// TIA Portal V15.1 export
// export: Created 2024-05-17T05:38:38.2002518Z, ExportSetting WithDefaults, DisplayName Totally Integrated Automation Portal, DisplayVersion V15.1 Update 5, DisplayName TIA Portal Openness, DisplayVersion V15.1 Update 5, DisplayName SINAMICS Startdrive Advanced, DisplayVersion V15.1, DisplayName G130, G150, S120, S150, SINAMICS MV, S210, DisplayVersion V15.1, DisplayName G110M, G120, G120C, G120D, G120P, DisplayVersion V15.1, DisplayName STEP 7 Professional, DisplayVersion V15.1 Update 5, DisplayName STEP 7 Safety, DisplayVersion V15.1, DisplayName WinCC Professional, DisplayVersion V15.1 Update 5, DisplayName SIMATIC Visualization Architect, DisplayVersion V15.1
FUNCTION_BLOCK "LGBMotor2W1S-C"   // FB6612, FBD
TITLE = LGBMotor2W1S-C
{ S7_Optimized_Access := 'TRUE' }
AUTHOR : VCC
FAMILY : Actuator
VERSION : 0.1
// ============================================================================
// This "Motor-2Way-1Speed-Contactor" module is used in Applications when a Motor 
// 2 way - 1 speed equipped with contactors is needed.
// The module contains: a Motor loop equipped with 
// "1 Motor protection.
// "2 contactors (Set & Reset).
// "1 safety switch
// ============================================================================
// stored: AutoNumber false, IsIECCheckEnabled false, IsRetainMemResEnabled false, MemoryReserve 100, SetENOAutomatically False, UDAEnableTagReadback false
   VAR_INPUT
      I_EnableAlarm { ExternalAccessible := 'False'; ExternalVisible := 'False'; ExternalWritable := 'False'} : Bool;   // Enable Alarm
      I_MotorProtection { ExternalAccessible := 'False'; ExternalVisible := 'False'; ExternalWritable := 'False'} : Bool;   // Motor protection
      I_BrakeProtection { ExternalAccessible := 'False'; ExternalVisible := 'False'; ExternalWritable := 'False'} : Bool;   // Brake protection
      I_SafetySwitch { ExternalAccessible := 'False'; ExternalVisible := 'False'; ExternalWritable := 'False'} : Bool;   // Safety Switch
      I_SetMotorCmd { ExternalAccessible := 'False'; ExternalVisible := 'False'; ExternalWritable := 'False'} : Bool;   // Set Command from function after Interlock
      I_ResetMotorCmd { ExternalAccessible := 'False'; ExternalVisible := 'False'; ExternalWritable := 'False'} : Bool;   // Reset Command from function after Interlock
      I_AlarmResetPB { ExternalAccessible := 'False'; ExternalVisible := 'False'; ExternalWritable := 'False'} : Bool;   // Alarm Reset Pushbutton is Activated
      I_SafetyOk { ExternalAccessible := 'False'; ExternalVisible := 'False'; ExternalWritable := 'False'} : Bool;   // Safety Ok
      I_MotionStopOk { ExternalAccessible := 'False'; ExternalVisible := 'False'; ExternalWritable := 'False'} : Bool;   // Safety Ok / The motion stop is Ok
      I_BrakeReleased { ExternalAccessible := 'False'; ExternalVisible := 'False'; ExternalWritable := 'False'} : Bool;   // Brake Released or not used
   END_VAR
   VAR_OUTPUT
      O_MotorProtectionAlm { ExternalAccessible := 'False'; ExternalVisible := 'False'; ExternalWritable := 'False'} : Bool;   // Motor protection Alarm
      O_BrakeProtectionAlm { ExternalAccessible := 'False'; ExternalVisible := 'False'; ExternalWritable := 'False'} : Bool;   // Brake protection alarm
      O_SafetySwitchAlm { ExternalAccessible := 'False'; ExternalVisible := 'False'; ExternalWritable := 'False'} : Bool;   // Safety Switch Alarm
      O_MotionStopWarning { ExternalAccessible := 'False'; ExternalVisible := 'False'; ExternalWritable := 'False'} : Bool;   // Drive fault / Motion Stop warning
      O_BrakeFeedbackAlm { ExternalAccessible := 'False'; ExternalVisible := 'False'; ExternalWritable := 'False'} : Bool;   // Brake Feedback Alm
      O_SetContactor { ExternalAccessible := 'False'; ExternalVisible := 'False'; ExternalWritable := 'False'} : Bool;   // Set Contactor of Motor loop
      O_ResetContactor { ExternalAccessible := 'False'; ExternalVisible := 'False'; ExternalWritable := 'False'} : Bool;   // Reset Contactor of Motor loop
      O_ReleaseBrake { ExternalAccessible := 'False'; ExternalVisible := 'False'; ExternalWritable := 'False'} : Bool;   // Release Brake Contactor
      O_AlarmABCondition { ExternalAccessible := 'False'; ExternalVisible := 'False'; ExternalWritable := 'False'} : Bool;   // Alarm AB Condition
      O_Active { ExternalAccessible := 'False'; ExternalVisible := 'False'; ExternalWritable := 'False'} : Bool;   // Motor loop Active
   END_VAR
   VAR_IN_OUT
      IO_Modes : "Modes";
      IO_Alarm : "Alarm";
      H_HMI : "H_HMI";
      "H_GBMotor2W1S-C" : "H_GBMotor2W1S-C";   // Animation
      C_SafetySwNc { ExternalAccessible := 'False'; ExternalVisible := 'False'; ExternalWritable := 'False'} : Bool;   // Safety switch Normally closed
      C_SafetySwitchUsed { ExternalAccessible := 'False'; ExternalVisible := 'False'; ExternalWritable := 'False'} : Bool;   // Safety switch used
      C_MotorProtectionNc { ExternalAccessible := 'False'; ExternalVisible := 'False'; ExternalWritable := 'False'} : Bool;   // Motor Protection Normally closed
      C_MotorProtectionUsed { ExternalAccessible := 'False'; ExternalVisible := 'False'; ExternalWritable := 'False'} : Bool;   // Motor Protection used
      C_BrakeProtectionNc { ExternalAccessible := 'False'; ExternalVisible := 'False'; ExternalWritable := 'False'} : Bool;   // Motor Protection Normally closed / Brake Protection Normally closed
      C_BrakeProtectionUsed { ExternalAccessible := 'False'; ExternalVisible := 'False'; ExternalWritable := 'False'} : Bool;   // Brake Protection used / Motor Protection used
      C_BrakeUsed { ExternalAccessible := 'False'; ExternalVisible := 'False'; ExternalWritable := 'False'} : Bool;   // Brake Release Used
      C_MotionStopUsed { ExternalAccessible := 'False'; ExternalVisible := 'False'; ExternalWritable := 'False'} : Bool;   // Motion Stop used
   END_VAR
   VAR
      MotorProtectionAlm { ExternalAccessible := 'False'; ExternalVisible := 'False'; ExternalWritable := 'False'} : Bool;   // Motor protection Alarm
      BrakeProtectionAlm { ExternalAccessible := 'False'; ExternalVisible := 'False'; ExternalWritable := 'False'} : Bool;   // Brake protection alarm
      SafetySwitchAlm { ExternalAccessible := 'False'; ExternalVisible := 'False'; ExternalWritable := 'False'} : Bool;   // Safety Switch Alarm
      MotorProtectionAlmCond { ExternalAccessible := 'False'; ExternalVisible := 'False'; ExternalWritable := 'False'} : Bool;   // Motor protection Alarm condition
      BrakeProtectionAlmCond { ExternalAccessible := 'False'; ExternalVisible := 'False'; ExternalWritable := 'False'} : Bool;   // Brake protection alarm condition
      SafetySwitchAlmCond { ExternalAccessible := 'False'; ExternalVisible := 'False'; ExternalWritable := 'False'} : Bool;   // Safety Switch Alarm condition
      BrakeFeedbackAlm { ExternalAccessible := 'False'; ExternalVisible := 'False'; ExternalWritable := 'False'} : Bool;   // Safety Switch alarm / Safety Switch Alarm / BrakeFeedbackAlm
      MotionStopWarning { ExternalAccessible := 'False'; ExternalVisible := 'False'; ExternalWritable := 'False'} : Bool;   // Drive fault alarm / Motion Stop warning
      SetContactor { ExternalAccessible := 'False'; ExternalVisible := 'False'; ExternalWritable := 'False'} : Bool;   // Set Contactor of Motor loop
      ResetContactor { ExternalAccessible := 'False'; ExternalVisible := 'False'; ExternalWritable := 'False'} : Bool;   // Reset Contactor of Motor loop
      Active { ExternalAccessible := 'False'; ExternalVisible := 'False'; ExternalWritable := 'False'} : Bool;   // Motor loop Active
      _MotorProtection { ExternalAccessible := 'False'; ExternalVisible := 'False'; ExternalWritable := 'False'} : "L1AlarmMultiIn";   // FB
      _BrakeProtection { ExternalAccessible := 'False'; ExternalVisible := 'False'; ExternalWritable := 'False'} : "L1AlarmMultiIn";   // FB
      _SafetySwitch { ExternalAccessible := 'False'; ExternalVisible := 'False'; ExternalWritable := 'False'} : "L1AlarmMultiIn";   // FB
      _BrakeFeedback { ExternalAccessible := 'False'; ExternalVisible := 'False'; ExternalWritable := 'False'} : "L1AlarmMultiIn";   // FB
      _MotionStop { ExternalAccessible := 'False'; ExternalVisible := 'False'; ExternalWritable := 'False'} : "L1AlarmMultiIn";   // FB
      _TimeBrakeRelease { ExternalAccessible := 'False'; ExternalVisible := 'False'; ExternalWritable := 'False'} : TON_TIME;
      edge { ExternalAccessible := 'False'; ExternalVisible := 'False'; ExternalWritable := 'False'} : Array[0..1] of Bool;
   END_VAR
   VAR_TEMP   // added for the SCL form of the ladder/FBD networks
      _w1 : Bool;
      _w2 : Bool;
   END_VAR
BEGIN

REGION Network 1: ****2.1 - Enable Alarms **** Enable Brake Feedback Alarm
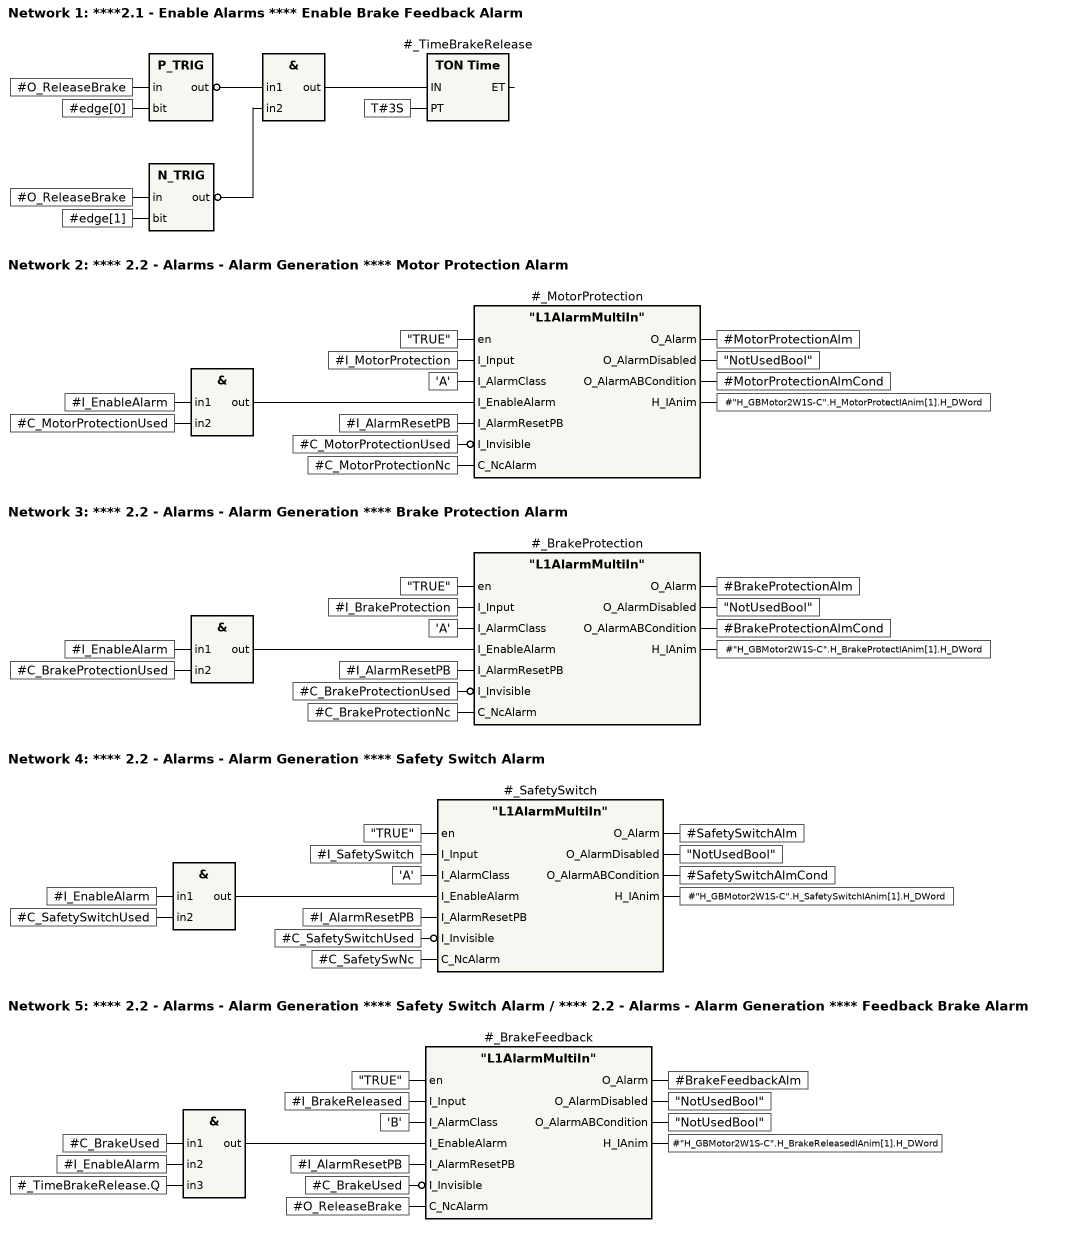
   #_w1 := #O_ReleaseBrake AND NOT #edge[0];   // rising edge
   #edge[0] := #O_ReleaseBrake;
   #_w2 := NOT #O_ReleaseBrake AND #edge[1];   // falling edge
   #edge[1] := #O_ReleaseBrake;
   #_TimeBrakeRelease(IN := NOT #_w1 AND NOT #_w2, PT := T#3S);   // TON
END_REGION

REGION Network 2: **** 2.2 - Alarms - Alarm Generation **** Motor Protection Alarm
   // Motor Protection Alarm
   IF "TRUE" THEN
       #_MotorProtection(I_Input := #I_MotorProtection,   // "L1AlarmMultiIn"
                         I_AlarmClass := 'A',
                         I_EnableAlarm := #I_EnableAlarm AND #C_MotorProtectionUsed,
                         I_AlarmResetPB := #I_AlarmResetPB,
                         I_Invisible := NOT #C_MotorProtectionUsed,
                         C_NcAlarm := #C_MotorProtectionNc,
                         O_Alarm => #MotorProtectionAlm,
                         O_AlarmDisabled => "NotUsedBool",
                         O_AlarmABCondition => #MotorProtectionAlmCond,
                         H_IAnim => #"H_GBMotor2W1S-C".H_MotorProtectIAnim[1].H_DWord);
   END_IF;
END_REGION

REGION Network 3: **** 2.2 - Alarms - Alarm Generation **** Brake Protection Alarm
   // Brake Protection Alarm
   IF "TRUE" THEN
       #_BrakeProtection(I_Input := #I_BrakeProtection,   // "L1AlarmMultiIn"
                         I_AlarmClass := 'A',
                         I_EnableAlarm := #I_EnableAlarm AND #C_BrakeProtectionUsed,
                         I_AlarmResetPB := #I_AlarmResetPB,
                         I_Invisible := NOT #C_BrakeProtectionUsed,
                         C_NcAlarm := #C_BrakeProtectionNc,
                         O_Alarm => #BrakeProtectionAlm,
                         O_AlarmDisabled => "NotUsedBool",
                         O_AlarmABCondition => #BrakeProtectionAlmCond,
                         H_IAnim => #"H_GBMotor2W1S-C".H_BrakeProtectIAnim[1].H_DWord);
   END_IF;
END_REGION

REGION Network 4: **** 2.2 - Alarms - Alarm Generation **** Safety Switch Alarm
   // Safety Switch Alarm
   IF "TRUE" THEN
       #_SafetySwitch(I_Input := #I_SafetySwitch,   // "L1AlarmMultiIn"
                      I_AlarmClass := 'A',
                      I_EnableAlarm := #I_EnableAlarm AND #C_SafetySwitchUsed,
                      I_AlarmResetPB := #I_AlarmResetPB,
                      I_Invisible := NOT #C_SafetySwitchUsed,
                      C_NcAlarm := #C_SafetySwNc,
                      O_Alarm => #SafetySwitchAlm,
                      O_AlarmDisabled => "NotUsedBool",
                      O_AlarmABCondition => #SafetySwitchAlmCond,
                      H_IAnim => #"H_GBMotor2W1S-C".H_SafetySwitchIAnim[1].H_DWord);
   END_IF;
END_REGION

REGION Network 5: **** 2.2 - Alarms - Alarm Generation **** Safety Switch Alarm / **** 2.2 - Alarms - Alarm Generation **** Feedback Brake Alarm
   // Safety Switch Alarm / Feedback Brake Alarm
   IF "TRUE" THEN
       #_BrakeFeedback(I_Input := #I_BrakeReleased,   // "L1AlarmMultiIn"
                       I_AlarmClass := 'B',
                       I_EnableAlarm := #C_BrakeUsed AND #I_EnableAlarm AND #_TimeBrakeRelease.Q,
                       I_AlarmResetPB := #I_AlarmResetPB,
                       I_Invisible := NOT #C_BrakeUsed,
                       C_NcAlarm := #O_ReleaseBrake,
                       O_Alarm => #BrakeFeedbackAlm,
                       O_AlarmDisabled => "NotUsedBool",
                       O_AlarmABCondition => "NotUsedBool",
                       H_IAnim => #"H_GBMotor2W1S-C".H_BrakeReleasedIAnim[1].H_DWord);
   END_IF;
END_REGION

REGION Network 6: **** 2.2 - Alarms - Alarm Generation **** MotionStop Warning
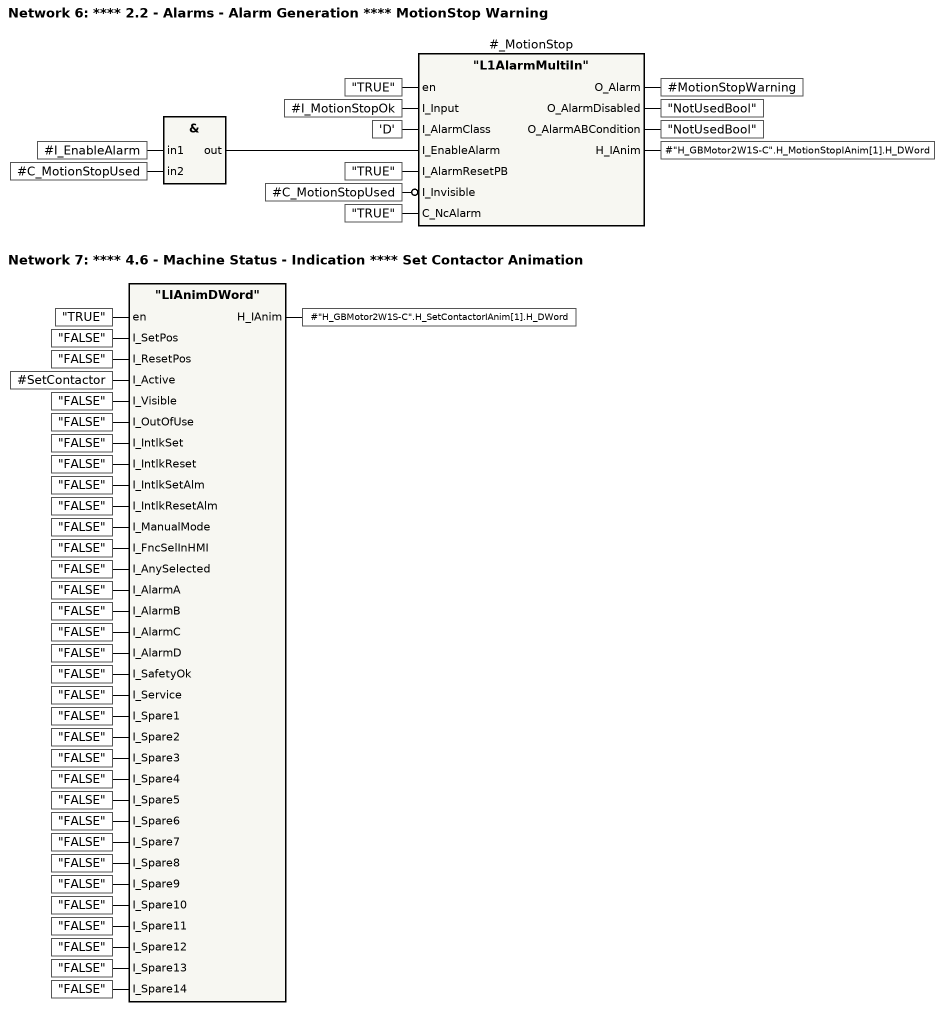
   IF "TRUE" THEN
       #_MotionStop(I_Input := #I_MotionStopOk,   // "L1AlarmMultiIn"
                    I_AlarmClass := 'D',
                    I_EnableAlarm := #I_EnableAlarm AND #C_MotionStopUsed,
                    I_AlarmResetPB := "TRUE",
                    I_Invisible := NOT #C_MotionStopUsed,
                    C_NcAlarm := "TRUE",
                    O_Alarm => #MotionStopWarning,
                    O_AlarmDisabled => "NotUsedBool",
                    O_AlarmABCondition => "NotUsedBool",
                    H_IAnim => #"H_GBMotor2W1S-C".H_MotionStopIAnim[1].H_DWord);
   END_IF;
END_REGION

REGION Network 7: **** 4.6 - Machine Status - Indication **** Set Contactor Animation
   // Set Contactor Animation
   IF "TRUE" THEN
       "LIAnimDWord"(I_SetPos := "FALSE",
                     I_ResetPos := "FALSE",
                     I_Active := #SetContactor,
                     I_Visible := "FALSE",
                     I_OutOfUse := "FALSE",
                     I_IntlkSet := "FALSE",
                     I_IntlkReset := "FALSE",
                     I_IntlkSetAlm := "FALSE",
                     I_IntlkResetAlm := "FALSE",
                     I_ManualMode := "FALSE",
                     I_FncSelInHMI := "FALSE",
                     I_AnySelected := "FALSE",
                     I_AlarmA := "FALSE",
                     I_AlarmB := "FALSE",
                     I_AlarmC := "FALSE",
                     I_AlarmD := "FALSE",
                     I_SafetyOk := "FALSE",
                     I_Service := "FALSE",
                     I_Spare1 := "FALSE",
                     I_Spare2 := "FALSE",
                     I_Spare3 := "FALSE",
                     I_Spare4 := "FALSE",
                     I_Spare5 := "FALSE",
                     I_Spare6 := "FALSE",
                     I_Spare7 := "FALSE",
                     I_Spare8 := "FALSE",
                     I_Spare9 := "FALSE",
                     I_Spare10 := "FALSE",
                     I_Spare11 := "FALSE",
                     I_Spare12 := "FALSE",
                     I_Spare13 := "FALSE",
                     I_Spare14 := "FALSE",
                     H_IAnim => #"H_GBMotor2W1S-C".H_SetContactorIAnim[1].H_DWord);
   END_IF;
END_REGION

REGION Network 8: **** 4.6 - Machine Status - Indication **** Reset Contactor Animation
   // Reset Contactor Animation
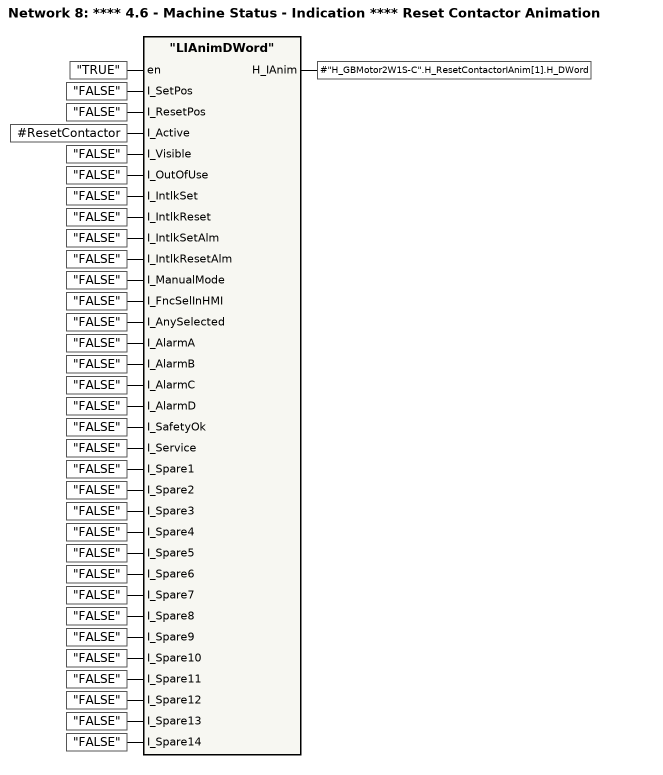
   IF "TRUE" THEN
       "LIAnimDWord"(I_SetPos := "FALSE",
                     I_ResetPos := "FALSE",
                     I_Active := #ResetContactor,
                     I_Visible := "FALSE",
                     I_OutOfUse := "FALSE",
                     I_IntlkSet := "FALSE",
                     I_IntlkReset := "FALSE",
                     I_IntlkSetAlm := "FALSE",
                     I_IntlkResetAlm := "FALSE",
                     I_ManualMode := "FALSE",
                     I_FncSelInHMI := "FALSE",
                     I_AnySelected := "FALSE",
                     I_AlarmA := "FALSE",
                     I_AlarmB := "FALSE",
                     I_AlarmC := "FALSE",
                     I_AlarmD := "FALSE",
                     I_SafetyOk := "FALSE",
                     I_Service := "FALSE",
                     I_Spare1 := "FALSE",
                     I_Spare2 := "FALSE",
                     I_Spare3 := "FALSE",
                     I_Spare4 := "FALSE",
                     I_Spare5 := "FALSE",
                     I_Spare6 := "FALSE",
                     I_Spare7 := "FALSE",
                     I_Spare8 := "FALSE",
                     I_Spare9 := "FALSE",
                     I_Spare10 := "FALSE",
                     I_Spare11 := "FALSE",
                     I_Spare12 := "FALSE",
                     I_Spare13 := "FALSE",
                     I_Spare14 := "FALSE",
                     H_IAnim => #"H_GBMotor2W1S-C".H_ResetContactorIAnim[1].H_DWord);
   END_IF;
END_REGION

REGION Network 9: **** 4.6 - Machine Status - Indication **** Reset Contactor Animation / **** 4.6 - Machine Status - Indication **** Release Brake Contactor Animation
   // Reset Contactor Animation
   // Release Brake Contactor Animation
   // Spare1 used to visualize the brake symbol on the contactor icon.
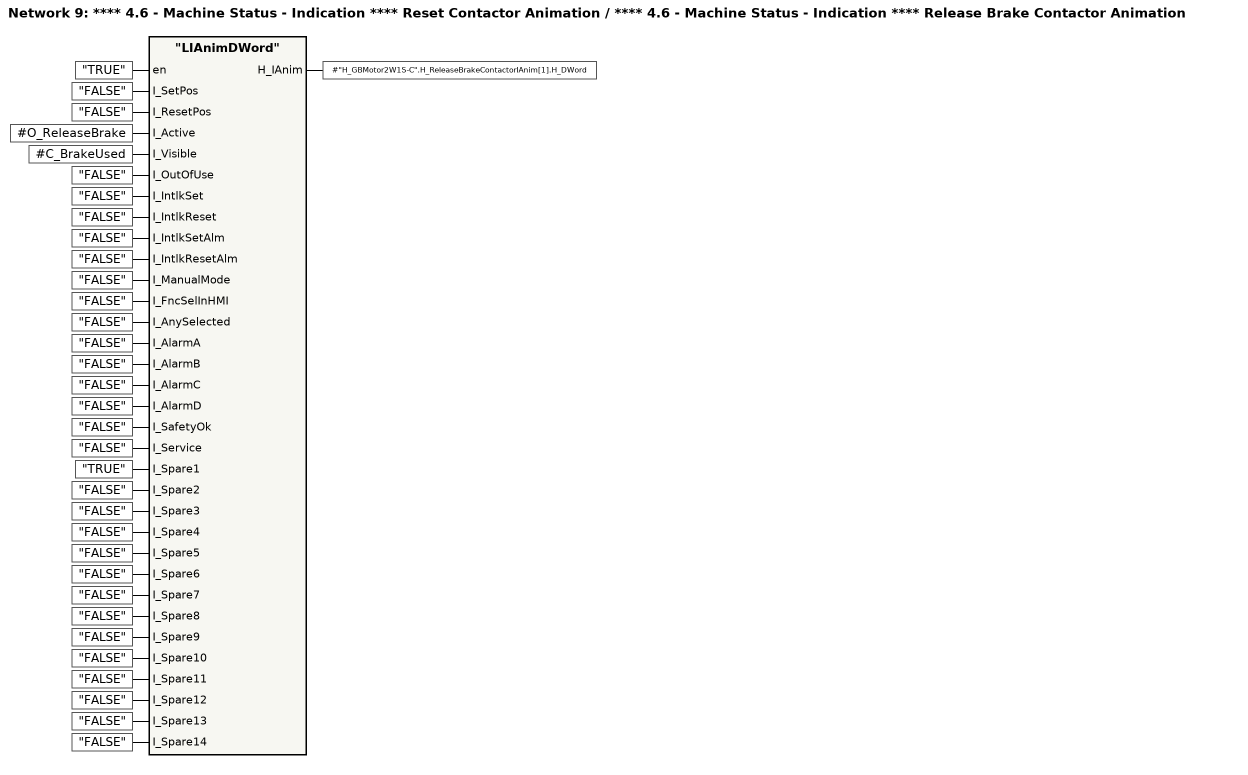
   IF "TRUE" THEN
       "LIAnimDWord"(I_SetPos := "FALSE",
                     I_ResetPos := "FALSE",
                     I_Active := #O_ReleaseBrake,
                     I_Visible := #C_BrakeUsed,
                     I_OutOfUse := "FALSE",
                     I_IntlkSet := "FALSE",
                     I_IntlkReset := "FALSE",
                     I_IntlkSetAlm := "FALSE",
                     I_IntlkResetAlm := "FALSE",
                     I_ManualMode := "FALSE",
                     I_FncSelInHMI := "FALSE",
                     I_AnySelected := "FALSE",
                     I_AlarmA := "FALSE",
                     I_AlarmB := "FALSE",
                     I_AlarmC := "FALSE",
                     I_AlarmD := "FALSE",
                     I_SafetyOk := "FALSE",
                     I_Service := "FALSE",
                     I_Spare1 := "TRUE",
                     I_Spare2 := "FALSE",
                     I_Spare3 := "FALSE",
                     I_Spare4 := "FALSE",
                     I_Spare5 := "FALSE",
                     I_Spare6 := "FALSE",
                     I_Spare7 := "FALSE",
                     I_Spare8 := "FALSE",
                     I_Spare9 := "FALSE",
                     I_Spare10 := "FALSE",
                     I_Spare11 := "FALSE",
                     I_Spare12 := "FALSE",
                     I_Spare13 := "FALSE",
                     I_Spare14 := "FALSE",
                     H_IAnim => #"H_GBMotor2W1S-C".H_ReleaseBrakeContactorIAnim[1].H_DWord);
   END_IF;
END_REGION

REGION Network 10: **** 4.6 - Machine Status - Indication **** Motor Icon Animation
   // Motor Animation
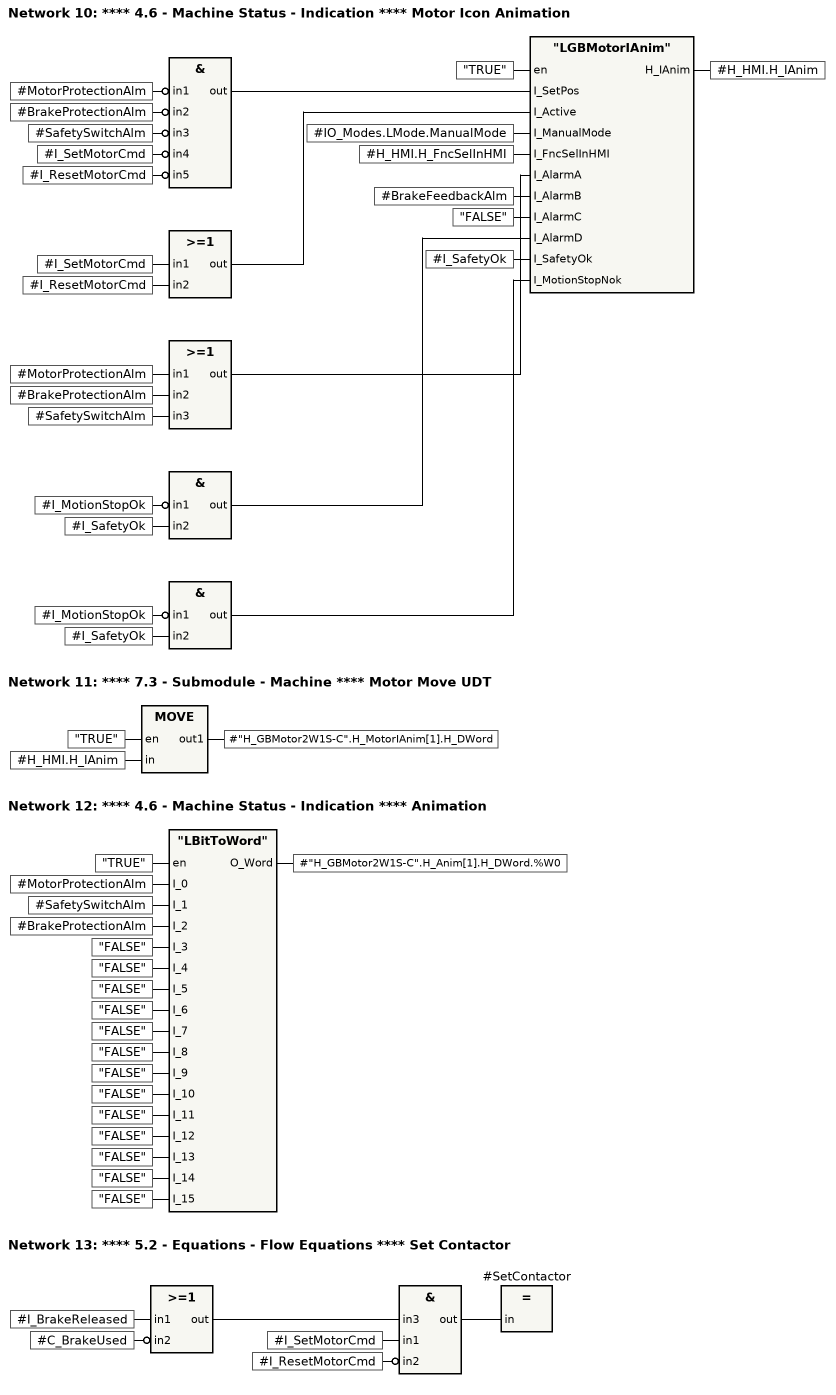
   IF "TRUE" THEN
       "LGBMotorIAnim"(I_SetPos := NOT #MotorProtectionAlm AND NOT #BrakeProtectionAlm AND NOT #SafetySwitchAlm AND NOT #I_SetMotorCmd AND NOT #I_ResetMotorCmd,
                       I_Active := #I_SetMotorCmd OR #I_ResetMotorCmd,
                       I_ManualMode := #IO_Modes.LMode.ManualMode,
                       I_FncSelInHMI := #H_HMI.H_FncSelInHMI,
                       I_AlarmA := #MotorProtectionAlm OR #BrakeProtectionAlm OR #SafetySwitchAlm,
                       I_AlarmB := #BrakeFeedbackAlm,
                       I_AlarmC := "FALSE",
                       I_AlarmD := NOT #I_MotionStopOk AND #I_SafetyOk,
                       I_SafetyOk := #I_SafetyOk,
                       I_MotionStopNok := NOT #I_MotionStopOk AND #I_SafetyOk,
                       H_IAnim => #H_HMI.H_IAnim);
   END_IF;
END_REGION

REGION Network 11: **** 7.3 - Submodule - Machine **** Motor Move UDT
   IF "TRUE" THEN #"H_GBMotor2W1S-C".H_MotorIAnim[1].H_DWord := #H_HMI.H_IAnim; END_IF;
END_REGION

REGION Network 12: **** 4.6 - Machine Status - Indication **** Animation
   // Animation
   IF "TRUE" THEN
       "LBitToWord"(I_0 := #MotorProtectionAlm,
                    I_1 := #SafetySwitchAlm,
                    I_2 := #BrakeProtectionAlm,
                    I_3 := "FALSE",
                    I_4 := "FALSE",
                    I_5 := "FALSE",
                    I_6 := "FALSE",
                    I_7 := "FALSE",
                    I_8 := "FALSE",
                    I_9 := "FALSE",
                    I_10 := "FALSE",
                    I_11 := "FALSE",
                    I_12 := "FALSE",
                    I_13 := "FALSE",
                    I_14 := "FALSE",
                    I_15 := "FALSE",
                    O_Word => #"H_GBMotor2W1S-C".H_Anim[1].H_DWord.%W0);
   END_IF;
END_REGION

REGION Network 13: **** 5.2 - Equations - Flow Equations **** Set Contactor
   // Set Contactor
   #SetContactor := (#I_BrakeReleased OR NOT #C_BrakeUsed) AND #I_SetMotorCmd AND NOT #I_ResetMotorCmd;
END_REGION

REGION Network 14: **** 5.2 - Equations - Flow Equations **** Reset Contactor
   // Reset Contactor
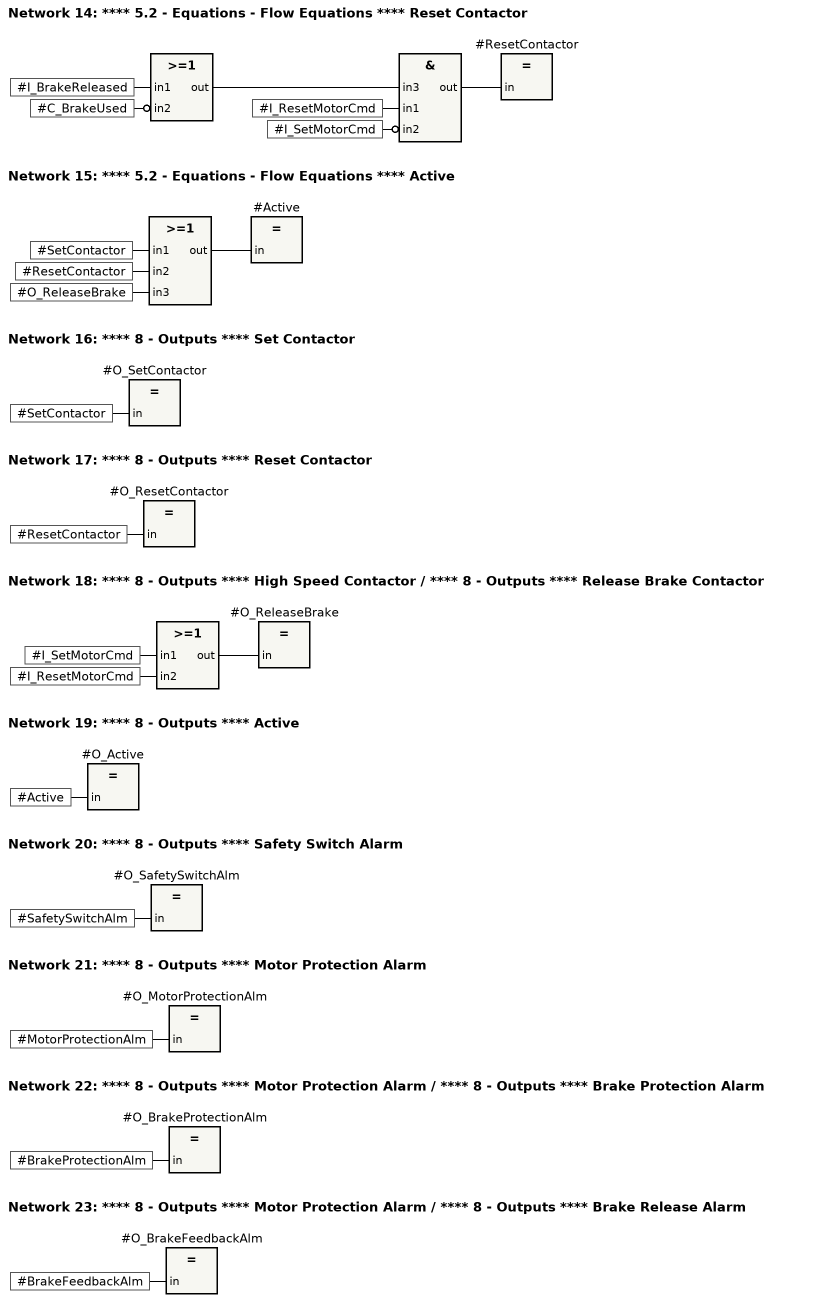
   #ResetContactor := (#I_BrakeReleased OR NOT #C_BrakeUsed) AND #I_ResetMotorCmd AND NOT #I_SetMotorCmd;
END_REGION

REGION Network 15: **** 5.2 - Equations - Flow Equations **** Active
   // Active
   #Active := #SetContactor OR #ResetContactor OR #O_ReleaseBrake;
END_REGION

REGION Network 16: **** 8 - Outputs **** Set Contactor
   // Set Contactor
   #O_SetContactor := #SetContactor;
END_REGION

REGION Network 17: **** 8 - Outputs **** Reset Contactor
   // Reset Contactor
   #O_ResetContactor := #ResetContactor;
END_REGION

REGION Network 18: **** 8 - Outputs **** High Speed Contactor / **** 8 - Outputs **** Release Brake Contactor
   // High Speed Contactor / Release Brake Contactor
   #O_ReleaseBrake := #I_SetMotorCmd OR #I_ResetMotorCmd;
END_REGION

REGION Network 19: **** 8 - Outputs **** Active
   // Active
   #O_Active := #Active;
END_REGION

REGION Network 20: **** 8 - Outputs **** Safety Switch Alarm
   // Safety Switch Alarm
   #O_SafetySwitchAlm := #SafetySwitchAlm;
END_REGION

REGION Network 21: **** 8 - Outputs **** Motor Protection Alarm
   // Motor Protection Alarm
   #O_MotorProtectionAlm := #MotorProtectionAlm;
END_REGION

REGION Network 22: **** 8 - Outputs **** Motor Protection Alarm / **** 8 - Outputs **** Brake Protection Alarm
   // Motor Protection Alarm / Brake Protection Alarm
   #O_BrakeProtectionAlm := #BrakeProtectionAlm;
END_REGION

REGION Network 23: **** 8 - Outputs **** Motor Protection Alarm / **** 8 - Outputs **** Brake Release Alarm
   // Motor Protection Alarm
   #O_BrakeFeedbackAlm := #BrakeFeedbackAlm;
END_REGION

REGION Network 24: **** 8 - Outputs **** Motion Stop warning
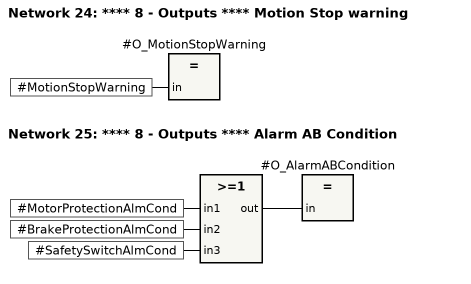
   #O_MotionStopWarning := #MotionStopWarning;
END_REGION

REGION Network 25: **** 8 - Outputs **** Alarm AB Condition
   // Alarm AB Condition
   #O_AlarmABCondition := #MotorProtectionAlmCond OR #BrakeProtectionAlmCond OR #SafetySwitchAlmCond;
END_REGION
END_FUNCTION_BLOCK
